// TwinCAT 3 PLC project Untitled1
// ProgramVersion: 3.1.4026.24
// libraries:
//   Tc2_Standard, * (Beckhoff Automation GmbH)
//   Tc2_System, * (Beckhoff Automation GmbH)
// project tree:
//   / PlcTask.TcTTO
//   POUs/ MAIN.TcPOU
// real-time tasks:
//   TASK PlcTask: cycle T#10ms, priority 20, ADS port 350

CONFIGURATION Untitled1
    RESOURCE PLC ON TwinCAT3
        TASK PlcTask(INTERVAL := T#10ms, PRIORITY := 20);
        PROGRAM MAIN WITH PlcTask : MAIN;
    END_RESOURCE
END_CONFIGURATION

// ---- POUs/MAIN.TcPOU
PROGRAM MAIN

VAR

bButton_1 	: BOOL	:=	FALSE; // INOUT SIGNAL FROM BUTTON 1 
bLamp_1 		: BOOL	:=	FALSE; // OUTPUT SIGNAL

END_VAR

bLamp_1 := bButton_1;

END_PROGRAM
